// TIA Portal V16 program export: 0 tag tables, 0 data types, 0 data blocks, 4 code blocks (in call order from the OBs), 0 instance data blocks

ORGANIZATION_BLOCK "Main"   // OB1, LAD, ProgramCycle
TITLE = "Main Program Sweep (Cycle)"
{ S7_Optimized_Access := 'TRUE' }
VERSION : 0.1
// stored: AutoNumber true, IsIECCheckEnabled false, SetENOAutomatically false
   VAR_INPUT
      Initial_Call : Bool;   // Initial call of this OB
      Remanence : Bool;   // =True, if remanent data are available
   END_VAR
   VAR_TEMP
      tTemp1 : Bool;
      tTemp2 : Bool;
   END_VAR
BEGIN

REGION Network 1: Komentarz
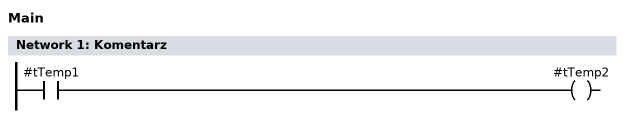
   RUNG wire#powerrail
      Contact( #tTemp1 )
      Coil( #tTemp2 )
   END_RUNG
   // the same network as SCL:
   #tTemp2 := #tTemp1;
END_REGION
END_ORGANIZATION_BLOCK

ORGANIZATION_BLOCK "qwe"   // OBqwe, LAD, ProgramCycle
TITLE = "Main Program Sweep (Cycle)"
{ S7_Optimized_Access := 'TRUE' }
VERSION : 0.1
// stored: AutoNumber true, IsIECCheckEnabled false, SetENOAutomatically false
   VAR_INPUT
      Initial_Call : Bool;   // Initial call of this OB
      qwe : Bool;   // =True, if remanent data are available
   END_VAR
   VAR_TEMP
      tTemp1 : Bool;
      tTemp2 : Bool;
   END_VAR
BEGIN

REGION Network 1: qwe
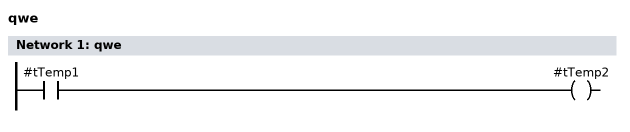
   RUNG wire#powerrail
      Contact( #tTemp1 )
      Coil( #tTemp2 )
   END_RUNG
   // the same network as SCL:
   #tTemp2 := #tTemp1;
END_REGION
END_ORGANIZATION_BLOCK

ORGANIZATION_BLOCK "$1"   // OB$2, LAD, ProgramCycle
TITLE = "Main Program Sweep (Cycle)"
{ S7_Optimized_Access := 'TRUE' }
VERSION : 0.1
// stored: AutoNumber true, IsIECCheckEnabled false, SetENOAutomatically false
   VAR_INPUT
      Initial_Call : Bool;   // Initial call of this OB
      "$6" : Bool;   // =True, if remanent data are available
   END_VAR
   VAR_TEMP
      tTemp1 : Bool;
      tTemp2 : Bool;
   END_VAR
BEGIN

REGION Network 1: $4
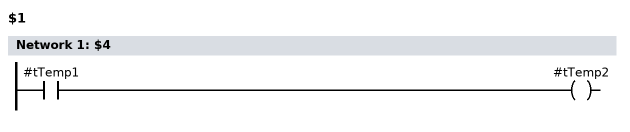
   RUNG wire#powerrail
      Contact( #tTemp1 )
      Coil( #tTemp2 )
   END_RUNG
   // the same network as SCL:
   #tTemp2 := #tTemp1;
END_REGION
END_ORGANIZATION_BLOCK

FUNCTION "funkcja1" : Void   // FC1, LAD
TITLE = taki oto jest tytuł bloku
{ S7_Optimized_Access := 'TRUE' }
VERSION : 0.1
// komentarz bloku
// stored: AutoNumber true, IsIECCheckEnabled false, SetENOAutomatically false, UDAEnableTagReadback false
BEGIN

REGION Network 1: komentarz linia 1
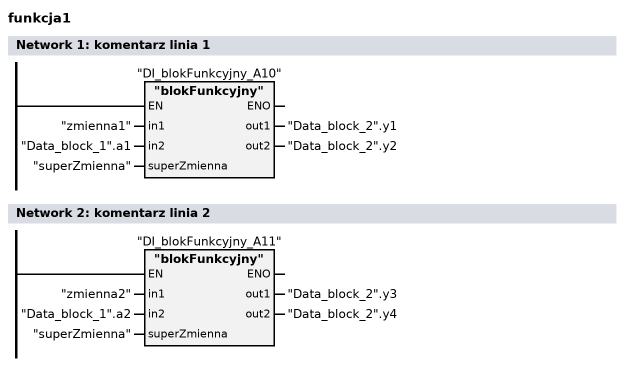
   RUNG wire#powerrail
      "DI_blokFunkcyjny_A10"(in1 := "zmienna1", in2 := "Data_block_1".a1, superZmienna := "superZmienna", out1 => "Data_block_2".y1, out2 => "Data_block_2".y2)
   END_RUNG
   // the same network as SCL:
   "DI_blokFunkcyjny_A10"(in1 := "zmienna1",   // "blokFunkcyjny"
                          in2 := "Data_block_1".a1,
                          superZmienna := "superZmienna",
                          out1 => "Data_block_2".y1,
                          out2 => "Data_block_2".y2);
END_REGION

REGION Network 2: komentarz linia 2
   RUNG wire#powerrail
      "DI_blokFunkcyjny_A11"(in1 := "zmienna2", in2 := "Data_block_1".a2, superZmienna := "superZmienna", out1 => "Data_block_2".y3, out2 => "Data_block_2".y4)
   END_RUNG
   // the same network as SCL:
   "DI_blokFunkcyjny_A11"(in1 := "zmienna2",   // "blokFunkcyjny"
                          in2 := "Data_block_1".a2,
                          superZmienna := "superZmienna",
                          out1 => "Data_block_2".y3,
                          out2 => "Data_block_2".y4);
END_REGION
END_FUNCTION
